### Operation Sequence
1. Validates that index is within valid range (0 to elementCount-1)
2. Validates that element size matches buffer element size (if element.diSize > 0)
3. Copies the element at the specified index to the output parameter
4. Shifts all elements after the index one position to the left using MEMMOVE
5. Clears the last position (now empty after the shift)
6. Decrements the element count

### Use Cases
```iecst
VAR
    buffer : AnyBuffer;
    value : DINT;
END_VAR

// Remove element from middle of buffer
buffer.PushRight(100);  // [100]
buffer.PushRight(200);  // [100, 200]
buffer.PushRight(300);  // [100, 200, 300]
buffer.PopAtIndex(1, value);  // value = 200, buffer = [100, 300]
```

### Performance Considerations
- **Time complexity**: O(n) - requires shifting elements after the index
- **Memory operations**: One memcpy for retrieval, one MEMMOVE for shifting, one memset for clearing
- **Cost varies by index**:
  - PopAtIndex(0) is equivalent to PopLeft - shifts all remaining elements
  - PopAtIndex(elementCount-1) is equivalent to PopRight - no shifting needed
  - Middle indices require partial shifting
- Use PopRight for O(1) removal when index doesn't matter
- Use for priority queues or sorted list maintenance

### Return Value
- **TRUE**: Element was successfully popped from the specified index
- **FALSE**: Pop operation failed (see error conditions)

### Error Conditions
- Returns FALSE and logs error if index is out of bounds (< 0 or >= elementCount)
- Returns FALSE and logs error if buffer is empty (elementCount = 0)
- Returns FALSE and logs error if element size doesn't match buffer element size (when element.diSize > 0)
- Element parameter can have diSize = 0 to discard the value without copying

### Side Effects
- Shifts all elements after the index one position to the left
- Clears the last element position (sets to zero)
- Decrements bufferMetadata.elementCount by 1

### Dependencies
- Uses memcpy for element retrieval
- Uses MEMMOVE for shifting elements (handles overlapping memory)
- Uses memset for clearing the last position
- Uses Trace for error logging

### Comparison with Other Methods
- **PopAtIndex(0)**: Same as PopLeft - removes from front, shifts all - O(n)
- **PopAtIndex(elementCount-1)**: Same as PopRight - removes from back, no shift - O(1)
- **PopAtIndex(middle)**: Removes from middle, shifts elements after index - O(n)
- **DeleteAtIndex**: Removes without retrieving value - O(1) for last index, O(n) otherwise

### Unittests
 - PopFromBeginning : verify popping at index 0 retrieves first element and shifts all
 - PopFromMiddle : verify popping from middle index retrieves correct element and shifts remaining
 - PopFromEnd : verify popping at last index (elementCount-1) retrieves last element
 - ReturnsTrueOnSuccess : verify method returns TRUE when pop succeeds
 - ReturnsFalseOnNegativeIndex : verify FALSE returned for negative index
 - ReturnsFalseOnIndexOutOfBounds : verify FALSE returned when index >= elementCount
 - ReturnsFalseOnEmptyBuffer : verify FALSE returned when buffer is empty (elementCount = 0)
 - WrongElementSize : verify FALSE returned when element size doesn't match
 - EmptyElement : verify behavior when element.diSize is 0 (discard mode)
 - ShiftsElementsCorrectly : verify all elements after index shift left by one position
 - ClearsLastPosition : verify the last position is cleared to zero after shift
 - DecrementsElementCount : verify elementCount decreases by 1 after pop
 - ConsecutivePops : verify multiple consecutive PopAtIndex calls maintain correct state
 - PopAllElements : verify can pop all elements sequentially using index 0
 - ElementOrderPreserved : verify element order is preserved after pop (except removed element)
 - PopAtIndexEquivalentToPopLeft : verify PopAtIndex(0) behaves same as PopLeft
 - PopAtIndexEquivalentToPopRight : verify PopAtIndex(elementCount-1) behaves same as PopRight
*)
PopAtIndex := FALSE;
// Check index bounds, cannot pop what is not filled in
IF index < bufferConfiguration.bufferBoundLower OR index >= bufferConfiguration.bufferBoundLower + bufferMetadata.elementCount THEN
	Trace.Error(__POUNAME(), CONCAT('Pop attempt at invalid index ', TO_STRING(index)));
	RETURN;
END_IF

// Check if buffer is empty
IF isEmpty THEN
	Trace.Error(__POUNAME(), 'Pop attempt on empty buffer');
	RETURN;
END_IF

// rebasedIndex necessary if LL <> 0
rebasedIndex := index - bufferConfiguration.bufferBoundLower;
// TRUE: passed type is not checked, element is discarded and not returned
IF NOT popDiscard THEN
	// Check element size if copy is requested (element.diSize > 0)
	IF element.diSize <> bufferConfiguration.elementSize THEN
		Trace.Error(__POUNAME(), CONCAT('Element size mismatch: expected ', CONCAT(TO_STRING(bufferConfiguration.elementSize), CONCAT(', got ', TO_STRING(element.diSize)))));
		RETURN;
	END_IF

	offset	 := rebasedIndex * bufferConfiguration.elementSize;
	destAddr := element.pValue;
	srcAddr	 := ADR(pBuffer.pValue[offset]);
	nBytes	 := TO_UDINT(element.diSize);
	memcpy(destAddr, srcAddr, nBytes);
END_IF

// Calculate how many elements need to be shifted
elementsToShift := bufferMetadata.elementCount - rebasedIndex - 1;
// Shift elements after the index one position to the left (if any)
IF elementsToShift > 0 THEN
	offset	 := rebasedIndex * bufferConfiguration.elementSize;
	destAddr := ADR(pBuffer.pValue[offset]);								   // destination: current index
	srcAddr	 := ADR(pBuffer.pValue[offset + bufferConfiguration.elementSize]); // source: next index
	nBytes	 := TO_UDINT(elementsToShift * bufferConfiguration.elementSize);
	MEMMOVE(destAddr, srcAddr, nBytes);
END_IF

// Delete last element data 
DeleteAtIndex(bufferMetadata.elementCount + bufferConfiguration.bufferBoundLower - 1);

// Update internal element counters 
CountDecrement();
PopAtIndex := TRUE;
END_METHOD

// Removes and retrieves the first element from the buffer (FIFO/queue operation)
METHOD PopLeft : BOOL
VAR_INPUT
	element	   : ANY;			// Variable to receive the popped element
	popDiscard : BOOL := FALSE; // When TRUE, element is removed but not copied (type checking skipped)
END_VAR

VAR
	offset	 : DINT;
	destAddr : PVOID;
	srcAddr	 : PVOID;
	nBytes	 : UDINT;
END_VAR

(*
## Detailed Description

Removes the first element from the left side of the buffer and optionally copies it to
the provided element parameter. This implements a standard FIFO (First-In-First-Out)
queue operation where elements are dequeued from the front.

The `popDiscard` parameter controls whether the removed element is copied to the output
parameter or simply discarded. This is useful for circular buffer scenarios where you need
to remove elements to make space without retrieving their values.

### Operation Sequence

**When popDiscard = FALSE (default - retrieve element):**
1. Validates that the buffer contains at least one element
2. Validates that element size matches the buffer's configured element size
3. Copies the first element to the output parameter
4. Shifts all remaining elements one position to the left
5. Clears the last position (now empty after the shift)
6. Decrements the element count

**When popDiscard = TRUE (discard element):**
1. Validates that the buffer contains at least one element
2. **Skips element size validation** (type checking bypassed)
3. **Skips copying element** to output parameter
4. Shifts all remaining elements one position to the left
5. Clears the last position (now empty after the shift)
6. Decrements the element count

### Parameters
- **element**: Variable to receive the popped element
  - When popDiscard=FALSE: Must match buffer's element size, receives the popped value
  - When popDiscard=TRUE: Can be any type/size, value is not copied (ignored)
- **popDiscard**: Controls whether to copy element or discard it
  - **FALSE (default)**: Element is validated and copied to output parameter
  - **TRUE**: Element validation is skipped, value is discarded (not copied)
  - Use TRUE for circular buffer overwrite scenarios where you don't need the old value

### Key Features
- **FIFO behavior**: Elements are removed in the order they were added (when combined with PushRight)
- **Optional discard mode**: Can remove element without retrieving it (popDiscard=TRUE)
- **Automatic shifting**: Maintains contiguous element storage after removal
- **Size validation**: Ensures the output element size matches buffer element size (when popDiscard=FALSE)
- **Type safety bypass**: popDiscard=TRUE skips type checking for performance in discard scenarios
- **Safe empty check**: Returns FALSE and logs error if buffer is empty

### Usage Example
```iecst
VAR
    queue : AnyBuffer(pBuffer := myBuffer, bufferBoundLower := 0, bufferBoundUpper := 9, isBufferPersistent := FALSE);
    value : DINT;
    discardBuffer : BYTE;  // Can be any type when using popDiscard=TRUE
    success : BOOL;
END_VAR

// Standard: Pop and retrieve the first element
success := queue.PopLeft(value, FALSE);  // or just queue.PopLeft(value)
IF success THEN
    // Process the retrieved value
END_IF

// Discard mode: Pop without retrieving (e.g., circular buffer overwrite)
success := queue.PopLeft(discardBuffer, TRUE);  // Element removed, value not copied
// OR with temporary pointer-based buffer:
pTemp := __NEW(BYTE, elementSize);
success := queue.PopLeft(pTemp^, TRUE);  // Element removed, discarded to temp buffer
__DELETE(pTemp);
```

### Performance Considerations
- **Time complexity**: O(n) due to element shifting (n = elementCount)
- **Memory operations**: Uses MEMMOVE for efficient bulk memory shifting
- **popDiscard=TRUE**: Slightly faster than popDiscard=FALSE (skips size check and memcpy)
- For frequent left-side operations, consider if a circular buffer would be more efficient

### Return Value
- **TRUE**: Element was successfully popped (and copied if popDiscard=FALSE)
- **FALSE**: Pop operation failed (see error conditions)

### Error Conditions
- Returns FALSE and logs error if buffer is empty (elementCount <= 0)
- Returns FALSE and logs error if element size doesn't match buffer element size **when popDiscard=FALSE**
- When popDiscard=TRUE, element size validation is skipped (no error for size mismatch)

### Dependencies
- Calls DeleteAtIndex to decrement element count and clear the vacated position
- Uses memcpy for element retrieval
- Uses MEMMOVE for shifting elements (handles overlapping memory correctly)
- Uses Trace for error logging

### Unittests
 - RetrievesFirstElement : verify the first element value is copied to output element when popDiscard=FALSE
 - ShiftsElements : verify all elements shift left by one position after pop
 - ClearsLastElement : verify the last position is cleared to zero after shift
 - DecrementsElementCount : verify elementCount decreases by 1 after pop
 - ReturnsTrueOnSuccess : verify method returns TRUE when pop succeeds
 - WrongSize : verify FALSE returned when element size differs from buffer element size (popDiscard=FALSE)
 - EmptyElement : verify behavior when element.diSize is 0 (discard mode, shift only)
 - PopFromEmptyBuffer : verify behavior when buffer has no elements (elementCount = 0)
 - PopSingleElement : verify popping when buffer contains exactly one element
 - ConsecutivePops : verify multiple sequential pops maintain correct order and state
 - PopAfterPushLeft : verify LIFO behavior with PushLeft and PopLeft
 - PopAfterPushRight : verify FIFO behavior with PushRight and PopLeft
 - PopUntilEmpty : verify popping all elements until buffer is empty
 - ElementOrderPreserved : verify remaining elements shift correctly and maintain relative order
 - PopDiscardTrue : verify element is removed but not copied when popDiscard=TRUE
 - PopDiscardTrueSkipsTypeCheck : verify no error when element size is wrong and popDiscard=TRUE
 - PopDiscardTrueShiftsElements : verify elements still shift correctly when popDiscard=TRUE
 - PopDiscardTrueDecrementsCount : verify elementCount decreases when popDiscard=TRUE
 - PopDiscardFalseRetrievesValue : verify element value is copied when popDiscard=FALSE (default)
 - PopDiscardFalseValidatesType : verify type checking occurs when popDiscard=FALSE
 - PopDiscardWithWrongTypeSucceeds : verify PopLeft with wrong type succeeds when popDiscard=TRUE
 - PopDiscardReturnsTrueOnSuccess : verify method returns TRUE when popDiscard=TRUE succeeds
*)
PopLeft := FALSE;
// Check if buffer has elements to pop
IF bufferMetadata.elementCount <= 0 THEN
	Trace.Error(__POUNAME(), 'Cannot pop from empty buffer');
	RETURN;
END_IF

// TRUE: passed type is not checked, element is discarded and not returned
IF NOT popDiscard THEN
	// Check element size if copy is requested (element.diSize > 0)
	IF element.diSize <> bufferConfiguration.elementSize THEN
		Trace.Error(__POUNAME(), CONCAT('Element size mismatch: expected ', CONCAT(TO_STRING(bufferConfiguration.elementSize), CONCAT(', got ', TO_STRING(element.diSize)))));
		RETURN;
	END_IF

	destAddr := element.pValue;
	srcAddr	 := pBuffer.pValue;
	nBytes	 := TO_UDINT(element.diSize);
	memcpy(destAddr, srcAddr, nBytes);
END_IF

// Shift elements to the left
offset	 := bufferConfiguration.elementSize;
destAddr := pBuffer.pValue;
srcAddr	 := ADR(pBuffer.pValue[offset]);
nBytes	 := TO_UDINT((bufferMetadata.elementCount - 1) * bufferConfiguration.elementSize);
MEMMOVE(destAddr, srcAddr, nBytes);

// Delete last element data 
DeleteAtIndex(bufferConfiguration.bufferBoundLower + bufferMetadata.elementCount - 1);

// Update internal element counters 
CountDecrement();
PopLeft := TRUE;
END_METHOD

// Removes and retrieves the last element from the buffer (stack pop operation)
METHOD PopRight : BOOL
VAR_INPUT
	element	   : ANY;			// Variable to receive the popped element
	popDiscard : BOOL := FALSE; // When TRUE, element is removed but not copied (type checking skipped)
END_VAR

VAR
	offset	 : DINT;
	destAddr : PVOID;
	srcAddr	 : PVOID;
	nBytes	 : UDINT;
END_VAR

(*
## Detailed Description

Removes the last element from the right side (back) of the buffer and optionally copies it to
the provided element parameter. This implements a standard stack pop operation where elements
are removed from the back, which can be combined with PushRight for LIFO (Last-In-First-Out)
behavior.

The `popDiscard` parameter controls whether the removed element is copied to the output
parameter or simply discarded. This is useful for circular buffer scenarios where you need
to remove elements to make space without retrieving their values.

### Operation Sequence

**When popDiscard = FALSE (default - retrieve element):**
1. Validates that the buffer contains at least one element
2. Validates that element size matches the buffer's configured element size
3. Copies the last element (at index elementCount-1) to the output parameter
4. Clears the last element position using DeleteAtIndex
5. Decrements the element count
6. No shifting of other elements required

**When popDiscard = TRUE (discard element):**
1. Validates that the buffer contains at least one element
2. **Skips element size validation** (type checking bypassed)
3. **Skips copying element** to output parameter
4. Clears the last element position using DeleteAtIndex
5. Decrements the element count
6. No shifting of other elements required

### Parameters
- **element**: Variable to receive the popped element
  - When popDiscard=FALSE: Must match buffer's element size, receives the popped value
  - When popDiscard=TRUE: Can be any type/size, value is not copied (ignored)
- **popDiscard**: Controls whether to copy element or discard it
  - **FALSE (default)**: Element is validated and copied to output parameter
  - **TRUE**: Element validation is skipped, value is discarded (not copied)
  - Use TRUE for circular buffer overwrite scenarios where you don't need the old value

### Key Features
- **LIFO behavior**: When combined with PushRight, provides stack behavior (last appended is first popped)
- **FIFO behavior**: When combined with PushLeft, provides queue behavior (first appended is last popped)
- **No shifting required**: Direct removal from the end without moving other elements
- **O(1) time complexity**: Constant time operation (much faster than PopLeft)
- **Optional discard mode**: Can remove element without retrieving it (popDiscard=TRUE)
- **Size validation**: Ensures the output element size matches buffer element size (when popDiscard=FALSE)
- **Type safety bypass**: popDiscard=TRUE skips type checking for performance in discard scenarios
- **Safe empty check**: Returns FALSE and logs error if buffer is empty

### Usage Example
```iecst
VAR
    stack : AnyBuffer(pBuffer := myBuffer, bufferBoundLower := 0, bufferBoundUpper := 9, isBufferPersistent := FALSE);
    value : DINT;
    discardBuffer : BYTE;  // Can be any type when using popDiscard=TRUE
    success : BOOL;
END_VAR

// Standard: Pop and retrieve the last element
success := stack.PopRight(value, FALSE);  // or just stack.PopRight(value)
IF success THEN
    // Process the retrieved value
END_IF

// Discard mode: Pop without retrieving (e.g., circular buffer overwrite)
success := stack.PopRight(discardBuffer, TRUE);  // Element removed, value not copied

// LIFO pattern: Last appended is first popped
stack.PushRight(1);  // [1]
stack.PushRight(2);  // [1, 2]
stack.PushRight(3);  // [1, 2, 3]
stack.PopRight(value); // value = 3, buffer = [1, 2]
```

### Performance Considerations
- **Time complexity**: O(1) - constant time operation (no shifting required)
- **Memory operations**: Single memcpy for element retrieval (when popDiscard=FALSE), memset for clearing
- **popDiscard=TRUE**: Slightly faster than popDiscard=FALSE (skips size check and memcpy)
- **Optimal for stack operations**: Use PushRight + PopRight for efficient LIFO stack
- Much faster than PopLeft since no element shifting is needed
- Preferred method for stack-based data structures

### Return Value
- **TRUE**: Element was successfully popped (and copied if popDiscard=FALSE)
- **FALSE**: Pop operation failed (see error conditions)

### Error Conditions
- Returns FALSE and logs error if buffer is empty (elementCount <= 0)
- Returns FALSE and logs error if element size doesn't match buffer element size **when popDiscard=FALSE**
- When popDiscard=TRUE, element size validation is skipped (no error for size mismatch)

### Side Effects
- Clears the last element position (sets to zero)
- Decrements bufferMetadata.elementCount by 1
- No other elements are moved or modified

### Dependencies
- Calls DeleteAtIndex to decrement element count and clear the position
- Uses memcpy for element retrieval
- Uses Trace for error logging

### Comparison with Other Methods
- **PopRight**: Removes from back (index elementCount-1), no shifting - O(1)
- **PopLeft**: Removes from front (index 0), shifts left - O(n)
- **PushRight**: Adds at back, no shifting - O(1)
- **PushLeft**: Adds at front, shifts right - O(n)

### Unittests
 - RetrievesLastElement : verify the last element value is copied to output element when popDiscard=FALSE
 - DoesNotShiftElements : verify no elements are shifted after pop
 - ClearsLastElement : verify the last position is cleared to zero after pop
 - DecrementsElementCount : verify elementCount decreases by 1 after pop
 - ReturnsTrueOnSuccess : verify method returns TRUE when pop succeeds
 - WrongSize : verify FALSE returned when element size differs from buffer element size (popDiscard=FALSE)
 - EmptyElement : verify behavior when element.diSize is 0 (discard mode, no copy)
 - PopFromEmptyBuffer : verify behavior when buffer has no elements (elementCount = 0)
 - PopSingleElement : verify popping when buffer contains exactly one element
 - ConsecutivePops : verify multiple sequential pops maintain correct order and state
 - PopAfterPushRight : verify LIFO behavior with PushRight and PopRight
 - PopAfterPushLeft : verify FIFO behavior with PushLeft and PopRight
 - PopUntilEmpty : verify popping all elements until buffer is empty
 - ElementOrderPreserved : verify remaining elements stay in their original positions
 - PopDiscardTrue : verify element is removed but not copied when popDiscard=TRUE
 - PopDiscardTrueSkipsTypeCheck : verify no error when element size is wrong and popDiscard=TRUE
 - PopDiscardTrueNoShift : verify no element shifting occurs when popDiscard=TRUE (same as default)
 - PopDiscardTrueDecrementsCount : verify elementCount decreases when popDiscard=TRUE
 - PopDiscardFalseRetrievesValue : verify element value is copied when popDiscard=FALSE (default)
 - PopDiscardFalseValidatesType : verify type checking occurs when popDiscard=FALSE
 - PopDiscardWithWrongTypeSucceeds : verify PopRight with wrong type succeeds when popDiscard=TRUE
 - PopDiscardReturnsTrueOnSuccess : verify method returns TRUE when popDiscard=TRUE succeeds
*)
PopRight := FALSE;
// Check if buffer has elements to pop
IF bufferMetadata.elementCount <= 0 THEN
	Trace.Error(__POUNAME(), 'Cannot pop from empty buffer');
	RETURN;
END_IF

// TRUE: passed type is not checked, element is discarded and not returned
IF NOT popDiscard THEN
	// Check element size if copy is requested (element.diSize > 0)
	IF element.diSize <> bufferConfiguration.elementSize THEN
		Trace.Error(__POUNAME(), CONCAT('Element size mismatch: expected ', CONCAT(TO_STRING(bufferConfiguration.elementSize), CONCAT(', got ', TO_STRING(element.diSize)))));
		RETURN;
	END_IF

	// Calculate offset to last element (elementCount - 1)
	offset	 := (bufferMetadata.elementCount - 1) * bufferConfiguration.elementSize;
	destAddr := element.pValue;
	srcAddr	 := ADR(pBuffer.pValue[offset]);
	nBytes	 := TO_UDINT(element.diSize);
	memcpy(destAddr, srcAddr, nBytes);
END_IF

// Delete last element data 
DeleteAtIndex(bufferConfiguration.bufferBoundLower + bufferMetadata.elementCount - 1);

// Update internal element counters 
CountDecrement();
PopRight := TRUE;
END_METHOD

// Insert an element at a specific index, shifting remaining elements right
METHOD PushAtIndex : BOOL
VAR_INPUT
	index	: DINT;
	element : ANY;
END_VAR

VAR
	offset			: DINT;
	destAddr		: PVOID;
	srcAddr			: PVOID;
	nBytes			: UDINT;
	elementsToShift : DINT;
	rebasedIndex	: DINT;
END_VAR

(*
## Detailed Description

Inserts a new element at the specified index by shifting all elements from that index onward
one position to the right, then placing the new element at the specified position. This provides
random-access insertion capability, allowing elements to be added at any position in the buffer
while maintaining contiguous storage.

### Operation Sequence
1. Validates that the buffer has been properly initialized
2. Checks that the buffer has space available (elementCount < capacity)
3. Validates that index is within valid range (0 to elementCount, inclusive)
4. Validates that the element size matches the buffer's configured element size
5. Shifts all elements from index onward one position to the right using MEMMOVE
6. Copies the new element to the specified index position
7. Increments the element count

### Use Cases
```iecst
VAR
    buffer : AnyBuffer;
    value : DINT;
END_VAR

// Insert at various positions
buffer.PushRight(100);  // [100]
buffer.PushRight(300);  // [100, 300]

value := 200;
buffer.PushAtIndex(1, value);  // [100, 200, 300] - inserted 200 between 100 and 300

value := 50;
buffer.PushAtIndex(0, value);  // [50, 100, 200, 300] - inserted 50 at beginning

value := 400;
buffer.PushAtIndex(4, value);  // [50, 100, 200, 300, 400] - inserted 400 at end
```

### Performance Considerations
- **Time complexity**: O(n) - requires shifting elements after the index
- **Memory operations**: One MEMMOVE for shifting, one memcpy for insertion
- **Cost varies by index**:
  - PushAtIndex(0) is equivalent to PushLeft - shifts all elements
  - PushAtIndex(elementCount) is equivalent to PushRight - no shifting needed
  - Middle indices require partial shifting
- Use PushRight for O(1) insertion when order doesn't matter
- Use for maintaining sorted order or priority queue operations

### Return Value
- **TRUE**: Element was successfully inserted at the specified index
- **FALSE**: Insert operation failed (see error conditions)

### Error Conditions
- Returns FALSE and logs error if buffer is not initialized
- Returns FALSE and logs error if buffer is full (elementCount >= capacity)
- Returns FALSE and logs error if index is out of bounds (< 0 or > elementCount)
- Returns FALSE and logs error if element size doesn't match buffer element size
- Note: index = elementCount is valid (append at end)

### Side Effects
- Shifts all elements from index onward one position to the right
- Increments bufferMetadata.elementCount by 1
- New element is placed at the specified index
- All elements at index and beyond move to index+1, index+2, etc.

### Dependencies
- Requires buffer to be initialized via FB_init or Initialize method
- Uses memcpy for element copying
- Uses MEMMOVE for shifting elements (handles overlapping memory correctly)
- Uses Trace for error logging

### Comparison with Other Methods
- **PushAtIndex(0)**: Same as PushLeft - shifts all, adds at front - O(n)
- **PushAtIndex(elementCount)**: Same as PushRight - no shift, adds at end - O(1)
- **PushAtIndex(middle)**: Inserts at middle, shifts elements after index - O(n)
- **PushLeft**: Always inserts at 0 - O(n)
- **PushRight**: Always inserts at end - O(1)

### Unittests
 - InsertAtBeginning : verify inserting at index 0 shifts all elements and inserts at front
 - InsertInMiddle : verify inserting at middle index shifts remaining elements correctly
 - InsertAtEnd : verify inserting at index elementCount appends at end (like PushRight)
 - InsertIntoEmptyBuffer : verify inserting at index 0 in empty buffer works
 - ReturnsTrueOnSuccess : verify method returns TRUE when insert succeeds
 - ReturnsFalseOnNegativeIndex : verify FALSE returned for negative index
 - ReturnsFalseOnIndexOutOfBounds : verify FALSE returned when index > elementCount
 - ReturnsFalseOnFullBuffer : verify FALSE returned when buffer is at capacity
 - WrongElementSize : verify FALSE returned when element size doesn't match
 - IncrementsElementCount : verify elementCount increases by 1 after insert
 - ShiftsElementsCorrectly : verify all elements from index onward shift right by one
 - PreservesElementOrder : verify element order is preserved after insert
 - MultipleInsertions : verify sequential insertions at different indices work correctly
 - InsertAllValidPositions : verify can insert at every valid position (0 to elementCount)
 - PushAtIndexEquivalentToPushLeft : verify PushAtIndex(0) behaves same as PushLeft
 - PushAtIndexEquivalentToPushRight : verify PushAtIndex(elementCount) behaves same as PushRight
*)
PushAtIndex := FALSE;
// Check if buffer has space available
IF isFull THEN
	Trace.Error(__POUNAME(), 'Cannot insert into full buffer');
	RETURN;
END_IF

// Check index bounds (0 to elementCount is valid - can insert at end)
IF index < bufferConfiguration.bufferBoundLower OR index > bufferConfiguration.bufferBoundLower + bufferMetadata.elementCount THEN
	Trace.Error(__POUNAME(), CONCAT('Insert attempt at invalid index ', TO_STRING(index)));
	RETURN;
END_IF

// Check if buffer is initialized
IF NOT isInitialized THEN
	Trace.Error(__POUNAME(), 'Buffer was not properly initialized before inserting');
	RETURN;
END_IF

// Validate element size matches buffer element size
IF element.diSize <> bufferConfiguration.elementSize THEN
	Trace.Error(__POUNAME(), 'Passed element to insert is of improper size');
	RETURN;
END_IF

// rebasedIndex necessary if LL <> 0
rebasedIndex := index - bufferConfiguration.bufferBoundLower;

// Calculate how many elements need to be shifted
elementsToShift := bufferMetadata.elementCount - rebasedIndex;
// Shift elements from index onward one position to the right (if any)
IF elementsToShift > 0 THEN
	offset	 := rebasedIndex * bufferConfiguration.elementSize;
	destAddr := ADR(pBuffer.pValue[offset + bufferConfiguration.elementSize]); // destination: index+1
	srcAddr	 := ADR(pBuffer.pValue[offset]);								   // source: current index
	nBytes	 := TO_UDINT(elementsToShift * bufferConfiguration.elementSize);
	MEMMOVE(destAddr, srcAddr, nBytes);
END_IF

// Copy the new element to the specified index position
offset	 := rebasedIndex * bufferConfiguration.elementSize;
destAddr := ADR(pBuffer.pValue[offset]);
srcAddr	 := element.pValue;
nBytes	 := TO_UDINT(element.diSize);
memcpy(destAddr, srcAddr, nBytes);

// Update internal element counters 
CountIncrement();
PushAtIndex := TRUE;
END_METHOD

// Appends a new element to the left side of the buffer (LIFO/stack push operation)
METHOD PushLeft : BOOL
VAR_INPUT
	element : ANY;
END_VAR

VAR
	offset	 : DINT;
	destAddr : PVOID;
	srcAddr	 : PVOID;
	nBytes	 : UDINT;
END_VAR

(*
## Detailed Description

Appends a new element to the left side (front) of the buffer by shifting all existing
elements one position to the right and inserting the new element at position 0. This
implements a stack-like push operation at the front, which can be combined with PopLeft
for LIFO (Last-In-First-Out) behavior.

### Operation Sequence
1. Validates that the buffer has been properly initialized
2. Checks that the buffer has space available (elementCount < capacity)
3. Validates that the element size matches the buffer's configured element size
4. Shifts all existing elements one position to the right using MEMMOVE
5. Copies the new element to position 0 (leftmost position)
6. Increments the element count

### Key Features
- **LIFO capability**: When combined with PopLeft, provides stack behavior (last appended is first popped)
- **FIFO capability**: When combined with PopRight, provides queue behavior (first appended is last popped)
- **Automatic shifting**: Maintains element contiguity by shifting existing elements right
- **Size validation**: Ensures the input element size matches buffer element size
- **Capacity checking**: Prevents buffer overflow by validating available space
- **Safe operation**: Validates initialization and capacity before modification

### Usage Example
```iecst
VAR
    stack : AnyBuffer(pBuffer := myBuffer, bufferBoundLower := 0, bufferBoundUpper := 9, isBufferPersistent := FALSE);
    value : DINT := 42;
    success : BOOL;
END_VAR

// Append element to the left (front)
success := stack.PushLeft(value);
IF success THEN
    // Element is now at position 0
    // All previous elements shifted right by one position
END_IF

// LIFO pattern: Last appended is first popped
stack.PushLeft(1);  // [1]
stack.PushLeft(2);  // [2, 1]
stack.PushLeft(3);  // [3, 2, 1]
stack.PopLeft(value); // value = 3, buffer = [2, 1]
```

### Performance Considerations
- **Time complexity**: O(n) due to element shifting (n = elementCount)
- **Memory operations**: Uses MEMMOVE for efficient bulk memory shifting
- **Shift overhead**: Every append requires shifting all existing elements
- For frequent left-side operations, consider if a circular buffer would be more efficient
- Use PopLeft with PushLeft for stack behavior (LIFO)
- Use PopRight with PushLeft for queue behavior (FIFO from right)

### Return Value
- **TRUE**: Element was successfully appended to the left side
- **FALSE**: Append operation failed (see error conditions)

### Error Conditions
- Returns FALSE and logs error if buffer is not initialized
- Returns FALSE and logs error if buffer is full (elementCount >= capacity)
- Returns FALSE and logs error if element size doesn't match buffer element size
- All errors are traced via the Trace system for debugging

### Side Effects
- Shifts all existing elements one position to the right
- Increments bufferMetadata.elementCount by 1
- New element is placed at index 0 (leftmost position)
- Previous element at index 0 moves to index 1, etc.

### Dependencies
- Requires buffer to be initialized via FB_init or Initialize method
- Uses memcpy for element copying
- Uses MEMMOVE for shifting elements (handles overlapping memory correctly)
- Uses Trace for error logging

### Comparison with Other Methods
- **PushLeft**: Adds at front (index 0), shifts right - O(n)
- **PopLeft**: Removes from front, shifts left - O(n)
- **PopRight**: Removes from back, no shifting - O(1)
- **PushAtIndex**: Adds at specific position - O(n)

### Unittests
 - AppendsToEmptyBuffer : verify element is inserted at position 0 in empty buffer
 - AppendsToNonEmptyBuffer : verify element is inserted at position 0 and existing elements shift right
 - IncrementsElementCount : verify elementCount increases by 1 after append
 - ShiftsExistingElements : verify all existing elements shift right by one position
 - ReturnsTrueOnSuccess : verify method returns TRUE when append succeeds
 - ReturnsFalseOnFullBuffer : verify method returns FALSE when buffer is at capacity
 - ReturnsFalseOnWrongSize : verify FALSE returned when element size doesn't match buffer element size
 - PreservesExistingData : verify existing element values remain unchanged after shift
 - AppendMultipleElements : verify consecutive appends work correctly (LIFO order)
 - AppendToFullBufferMinus1 : verify append succeeds when buffer has exactly 1 space remaining
 - AppendWhenFullCapacity : verify append fails when elementCount equals capacity
 - AppendZeroSizedElement : verify behavior when element.diSize is 0
 - AppendWithDifferentDataTypes : verify append works with various data types (DINT, REAL, struct)
 - ConsecutivePushAndPopLeft : verify LIFO behavior with alternating PushLeft and PopLeft calls
 - ConsecutivePushAndPopRight : verify FIFO behavior with alternating PushLeft and PopRight calls
 - ElementOrderAfterMultipleAppends : verify element order is correct after multiple appends
 - FillBufferCompletely : verify filling buffer to full capacity works correctly
*)
PushLeft := FALSE;
// Check if buffer has space available
IF isFull THEN
	Trace.Error(__POUNAME(), 'Cannot append to full buffer');
	RETURN;
END_IF

// Check if buffer is initialized
IF NOT isInitialized THEN
	Trace.Error(__POUNAME(), 'Buffer was not properly initialized before appending');
	RETURN;
END_IF

// Check element size if copy is requested (element.diSize > 0)
IF element.diSize <> bufferConfiguration.elementSize THEN
	Trace.Error(__POUNAME(), CONCAT('Element size mismatch: expected ', CONCAT(TO_STRING(bufferConfiguration.elementSize), CONCAT(', got ', TO_STRING(element.diSize)))));
	RETURN;
END_IF

// Shift all existing elements to the right to make room at position 0
destAddr := ADR(pBuffer.pValue[bufferConfiguration.elementSize]); // Start at position 1
srcAddr	 := pBuffer.pValue;										  // Start at position 0
nBytes	 := TO_UDINT(bufferMetadata.elementCount * bufferConfiguration.elementSize);
MEMMOVE(destAddr, srcAddr, nBytes);

// Copy the new element to position 0 (leftmost position)
destAddr := pBuffer.pValue;
srcAddr	 := element.pValue;
nBytes	 := TO_UDINT(element.diSize);
memcpy(destAddr, srcAddr, nBytes);

// Update internal element counters 
CountIncrement();
PushLeft := TRUE;
END_METHOD

// Appends a new element to the right side of the buffer (FIFO/queue enqueue operation)
METHOD PushRight : BOOL
VAR_INPUT
	element : ANY;
END_VAR

VAR
	offset	 : DINT;
	destAddr : PVOID;
	srcAddr	 : PVOID;
	nBytes	 : UDINT;
END_VAR

(*
## Detailed Description

Appends a new element to the right side (back) of the buffer by placing the element at
the next available position (index = elementCount). This implements a standard queue
enqueue operation where elements are added to the back, which can be combined with PopLeft
for FIFO (First-In-First-Out) behavior.

### Operation Sequence
1. Validates that the buffer has been properly initialized
2. Checks that the buffer has space available (elementCount < capacity)
3. Validates that the element size matches the buffer's configured element size
4. Copies the new element to position elementCount (rightmost available position)
5. Increments the element count

### Key Features
- **FIFO capability**: When combined with PopLeft, provides queue behavior (first appended is first popped)
- **LIFO capability**: When combined with PopRight, provides stack behavior (last appended is first popped)
- **No shifting required**: Direct placement at the end without moving existing elements
- **Size validation**: Ensures the input element size matches buffer element size
- **Capacity checking**: Prevents buffer overflow by validating available space
- **Safe operation**: Validates initialization and capacity before modification

### Usage Example
```iecst
VAR
    queue : AnyBuffer(pBuffer := myBuffer, bufferBoundLower := 0, bufferBoundUpper := 9, isBufferPersistent := FALSE);
    value : DINT := 42;
    success : BOOL;
END_VAR

// Append element to the right (back)
success := queue.PushRight(value);
IF success THEN
    // Element is now at position elementCount-1
    // No existing elements are moved
END_IF

// FIFO pattern: First appended is first popped
queue.PushRight(1);  // [1]
queue.PushRight(2);  // [1, 2]
queue.PushRight(3);  // [1, 2, 3]
queue.PopLeft(value);  // value = 1, buffer = [2, 3]
```

### Performance Considerations
- **Time complexity**: O(1) - constant time operation (no shifting required)
- **Memory operations**: Single memcpy for the new element
- **Optimal for queue operations**: Use PushRight + PopLeft for efficient FIFO queue
- Much faster than PushLeft since no element shifting is needed
- Preferred method for building up a buffer sequentially

### Return Value
- **TRUE**: Element was successfully appended to the right side
- **FALSE**: Append operation failed (see error conditions)

### Error Conditions
- Returns FALSE and logs error if buffer is not initialized
- Returns FALSE and logs error if buffer is full (elementCount >= capacity)
- Returns FALSE and logs error if element size doesn't match buffer element size
- All errors are traced via the Trace system for debugging

### Side Effects
- New element is placed at index elementCount (rightmost available position)
- Increments bufferMetadata.elementCount by 1
- No existing elements are moved or modified

### Dependencies
- Requires buffer to be initialized via FB_init or Initialize method
- Uses memcpy for element copying
- Uses Trace for error logging

### Comparison with Other Methods
- **PushRight**: Adds at back (index elementCount), no shifting - O(1)
- **PushLeft**: Adds at front (index 0), shifts right - O(n)
- **PopLeft**: Removes from front, shifts left - O(n)
- **PopRight**: Removes from back, no shifting - O(1)

### Unittests
 - AppendsToEmptyBuffer : verify element is inserted at position 0 in empty buffer
 - AppendsToNonEmptyBuffer : verify element is inserted at position elementCount and no elements shift
 - IncrementsElementCount : verify elementCount increases by 1 after append
 - DoesNotShiftElements : verify no existing elements are moved after append
 - ReturnsTrueOnSuccess : verify method returns TRUE when append succeeds
 - ReturnsFalseOnFullBuffer : verify method returns FALSE when buffer is at capacity
 - ReturnsFalseOnWrongSize : verify FALSE returned when element size doesn't match buffer element size
 - PreservesExistingData : verify existing element values remain unchanged
 - AppendMultipleElements : verify consecutive appends work correctly (FIFO order with PopLeft)
 - AppendToFullBufferMinus1 : verify append succeeds when buffer has exactly 1 space remaining
 - AppendWhenFullCapacity : verify append fails when elementCount equals capacity
 - AppendZeroSizedElement : verify behavior when element.diSize is 0
 - AppendWithDifferentDataTypes : verify append works with various data types (DINT, REAL, struct)
 - ConsecutivePushAndPopLeft : verify FIFO behavior with PushRight and PopLeft calls
 - ConsecutivePushAndPopRight : verify LIFO behavior with PushRight and PopRight calls
 - ElementOrderAfterMultipleAppends : verify element order is correct after multiple appends
 - FillBufferCompletely : verify filling buffer to full capacity works correctly
*)
PushRight := FALSE;
// Check if buffer has space available
IF isFull THEN
	Trace.Error(__POUNAME(), 'Cannot append to full buffer');
	RETURN;
END_IF

// Check if buffer is initialized
IF NOT isInitialized THEN
	Trace.Error(__POUNAME(), 'Buffer was not properly initialized before appending');
	RETURN;
END_IF

// Check element size if copy is requested (element.diSize > 0)
IF element.diSize <> bufferConfiguration.elementSize THEN
	Trace.Error(__POUNAME(), CONCAT('Element size mismatch: expected ', CONCAT(TO_STRING(bufferConfiguration.elementSize), CONCAT(', got ', TO_STRING(element.diSize)))));
	RETURN;
END_IF

// Copy the new element to position elementCount (rightmost available position)
offset	 := bufferMetadata.elementCount * bufferConfiguration.elementSize;
destAddr := ADR(pBuffer.pValue[offset]);
srcAddr	 := element.pValue;
nBytes	 := TO_UDINT(element.diSize);
memcpy(destAddr, srcAddr, nBytes);

// Update internal element counters 
CountIncrement();
PushRight := TRUE;
END_METHOD

// Overwrite an element at a specific index without changing buffer structure or the buffer counters
METHOD ReplaceAtIndex : BOOL
VAR_INPUT
	index	: DINT;
	element : ANY;
END_VAR

VAR
	offset		 : DINT;
	destAddr	 : PVOID;
	srcAddr		 : PVOID;
	nBytes		 : UDINT;
	rebasedIndex : DINT;
END_VAR

(*
## Detailed Description

Overwrites the element at the specified index with a new value without modifying the buffer
metadata or structure. This is a low-level primitive operation that replaces data in-place
without any shifting, insertion, deletion, or metadata updates. The caller is responsible
for validating buffer state if needed.

### Operation Sequence
1. Validates that index is within valid range (0 to capacity-1)
2. Validates that element size matches buffer element size (if element.diSize > 0)
3. Overwrites the element at the specified index with the new value
4. Returns without modifying element count or other elements

### Use Cases
```iecst
VAR
    buffer : AnyBuffer;
    value : DINT;
END_VAR

// Update specific positions (regardless of whether they're "filled")
value := 999;
buffer.ReplaceAtIndex(2, value);  // Overwrites position 2 with 999
// Works even if position 2 was not previously "filled" in logical sense
```

### Performance Considerations
- **Time complexity**: O(1) - constant time operation (direct indexed access)
- **Memory operations**: Single memcpy to overwrite element
- **No buffer modifications**: No shifting, no count changes, no state checking
- **In-place update**: Efficient for updating data at any buffer position
- Optimal for direct memory updates without overhead
- Use for low-level buffer manipulation or custom buffer management

### Return Value
- **TRUE**: Element was successfully replaced at the specified index
- **FALSE**: Replace operation failed (see error conditions)

### Error Conditions
- Returns FALSE and logs error if index is out of bounds (< 0 or >= capacity)
- Returns FALSE and logs error if element size doesn't match buffer element size (when element.diSize > 0)
- Element parameter can have diSize = 0 to skip replacement (returns TRUE if index valid)

### Side Effects
- **Minimal** - Only the element at the specified index is modified
- **Does NOT** modify elementCount or any other metadata
- **Does NOT** check if position is logically "filled" or if buffer is empty
- All other elements remain in their original positions with original values
- No memory allocation or deallocation

### Important Notes
- **No metadata changes**: Does NOT modify elementCount or validate buffer state
- **Caller responsibility**: Calling code must validate buffer state if needed
- **No state checking**: Works at any index within capacity, regardless of elementCount
- **Index range**: Valid indices are [0, capacity-1], not [0, elementCount-1]
- **Low-level primitive**: Designed for internal use or custom buffer management

### Dependencies
- Uses memcpy for element overwriting
- Uses Trace for error logging

### Comparison with Other Methods
- **ReplaceAtIndex**: Updates element at index - O(1), no metadata change
- **PopAtIndex**: Removes element at index - O(n), shifts and updates count
- **PeekAtIndex**: Reads element at index - O(1), validates elementCount
- **DeleteAtIndex**: Clears element - O(1), no metadata change

### Unittests
 - ReplaceAtBeginning : verify replacing at index 0 updates first element correctly
 - ReplaceInMiddle : verify replacing at middle index updates correct element
 - ReplaceAtEnd : verify replacing at last capacity index updates last element
 - ReturnsTrueOnSuccess : verify method returns TRUE when replace succeeds
 - ReturnsFalseOnNegativeIndex : verify FALSE returned for negative index
 - ReturnsFalseOnIndexAtCapacity : verify FALSE returned when index == capacity
 - ReturnsFalseOnIndexAboveCapacity : verify FALSE returned when index > capacity
 - WrongElementSize : verify FALSE returned when element size doesn't match
 - BufferUnchangedExceptIndex : verify all other elements remain unchanged after replace
 - MetadataUnchanged : verify elementCount and all metadata remain unchanged after replace
 - MultipleReplacements : verify sequential replacements at different indices work correctly
 - ReplaceAllCapacityPositions : verify can replace every capacity position (0 to capacity-1)
 - ReplaceWithDifferentValues : verify replace works with various data values
 - ReplaceSameIndexMultipleTimes : verify can overwrite same position repeatedly
 - ReplaceEmptyPosition : verify can replace position that was never filled (elementCount < index < capacity)
 - ReplaceWhenBufferEmpty : verify replace succeeds even when elementCount = 0 (if index < capacity)
*)
ReplaceAtIndex := FALSE;
// Check index bounds against capacity (caller manages state validation)
IF index < bufferConfiguration.bufferBoundLower OR index > bufferConfiguration.bufferBoundUpper THEN
	Trace.Error(__POUNAME(), CONCAT('Replace attempt at invalid index ', TO_STRING(index)));
	RETURN;
END_IF

// Check element size if copy is requested (element.diSize > 0)
IF element.diSize <> bufferConfiguration.elementSize THEN
	Trace.Error(__POUNAME(), CONCAT('Element size mismatch: expected ', CONCAT(TO_STRING(bufferConfiguration.elementSize), CONCAT(', got ', TO_STRING(element.diSize)))));
	RETURN;
END_IF

// rebasedIndex necessary if LL <> 0
rebasedIndex := index - bufferConfiguration.bufferBoundLower;

// Copy element at index to output parameter (if element.diSize > 0)
offset	 := rebasedIndex * bufferConfiguration.elementSize;
destAddr := ADR(pBuffer.pValue[offset]);
srcAddr	 := element.pValue;
nBytes	 := TO_UDINT(element.diSize);
memcpy(destAddr, srcAddr, nBytes);

// No buffer modifications - overwrite-only operation
ReplaceAtIndex := TRUE;
END_METHOD

END_FUNCTION_BLOCK

// Utilities/AnyBuffer/TypedBuffers/LifoBuffer
// Provides a simplified LIFO stack interface as an adapter over AnyBuffer
FUNCTION_BLOCK LifoBuffer IMPLEMENTS I_AnyBufferStrategy
VAR
	anyBuffer	  : I_AnyBuffer;
	isInitialized : BOOL := FALSE;
	_overwrite	  : BOOL := FALSE; // When TRUE, Push overwrites oldest element when full
	_reversed	  : BOOL := FALSE; // When TRUE, reverses push/pop direction (PushLeft/PopLeft)
	{attribute 'hide'}
	discardObject : BYTE; // element for discarding elements in overwrite mode
END_VAR

(*
## Detailed Description

LifoBuffer is an adapter (also known as a strategy or facade) that wraps an AnyBuffer instance
to provide a simplified Last-In-First-Out (LIFO) stack interface. Instead of using the full
AnyBuffer API with directional operations (PushLeft/Right, PopLeft/Right), users can simply
Push and Pop elements following standard stack semantics.

### Alternative Names
In computer science, LIFO data structures are commonly called "Stacks". This implementation
could alternatively be named "Stack" or "StackAdapter" for more conventional naming.

### Design Pattern
This implements the **Adapter Pattern** (also Strategy Pattern), which:
- Wraps a more complex interface (I_AnyBuffer) with a simpler, domain-specific interface
- Delegates all operations to the underlying AnyBuffer instance
- Provides semantic clarity: Push/Pop vs PushRight/PopRight
- Allows multiple strategy implementations (FIFO, LIFO, Priority, etc.) over the same buffer

### LIFO Semantics
- **Push(element)**: Adds element using PushRight (reversed=FALSE) or PushLeft (reversed=TRUE)
- **Pop(element)**: Removes element using PopRight (reversed=FALSE) or PopLeft (reversed=TRUE)
- Push and Pop operate on the **same end** of the buffer (unlike FIFO)
- Last element pushed is the first element popped (LIFO behavior)
- Elements maintain insertion order, but retrieval is in reverse order

### Configurable Behavior
The LifoBuffer supports two optional parameters during initialization:

**overwrite parameter:**
- **FALSE (default)**: Push fails when buffer is full, returns FALSE and logs error
- **TRUE**: Push to full buffer automatically removes element to make space (circular buffer behavior)
  - When reversed=FALSE: Removes from front (PopLeft), adds to back (PushRight)
  - When reversed=TRUE: Removes from back (PopRight), adds to front (PushLeft)
  - Removed element is discarded using internal temporary buffer

**reversed parameter:**
- **FALSE (default)**: Standard LIFO - Push to back (PushRight), Pop from back (PopRight)
- **TRUE**: Reversed direction - Push to front (PushLeft), Pop from front (PopLeft)
- Both Push and Pop operate on the **same end** to maintain LIFO semantics

### Operation Mapping
**Standard Mode (overwrite=FALSE, reversed=FALSE):**
```
Push()  -> anyBuffer.PushRight()  // Add to back (right)
Pop()   -> anyBuffer.PopRight()   // Remove from back (right) - LIFO
Clear() -> anyBuffer.Clear()      // Clear all
isEmpty -> anyBuffer.isEmpty      // Check if empty
isFull  -> anyBuffer.isFull       // Check if full
```

**Overwrite Mode (overwrite=TRUE, reversed=FALSE):**
```
Push()  -> if full: anyBuffer.PopLeft(pBufferTemp), then anyBuffer.PushRight()
Pop()   -> anyBuffer.PopRight()   // Remove from back (right)
```

**Reversed Mode (overwrite=FALSE, reversed=TRUE):**
```
Push()  -> anyBuffer.PushLeft()   // Add to front (left)
Pop()   -> anyBuffer.PopLeft()    // Remove from front (left) - LIFO
```

**Overwrite + Reversed Mode (overwrite=TRUE, reversed=TRUE):**
```
Push()  -> if full: anyBuffer.PopRight(pBufferTemp), then anyBuffer.PushLeft()
Pop()   -> anyBuffer.PopLeft()    // Remove from front (left)
```

### Usage Examples

**Standard LIFO Mode (Stack):**
```iecst
VAR
    rawBuffer : ARRAY[0..2] OF DINT;
    buffer : AnyBuffer(pBuffer := rawBuffer,
                       bufferBoundLower := 0,
                       bufferBoundUpper := 2,
                       isBufferPersistent := FALSE);
    lifo : LifoBuffer(anyBuffer := buffer, overwrite := FALSE, reversed := FALSE);
    value : DINT;
END_VAR

// Push elements (adds to back)
value := 100; lifo.Push(value);  // Stack: [100]
value := 200; lifo.Push(value);  // Stack: [100, 200] - 200 added to back
value := 300; lifo.Push(value);  // Stack: [100, 200, 300] - 300 added to back

// Pop elements (LIFO order - newest first)
lifo.Pop(value);   // value = 300 (from back), Stack: [100, 200]
lifo.Pop(value);   // value = 200 (from back), Stack: [100]
lifo.Pop(value);   // value = 100 (from back), Stack: []
```

**Overwrite Mode (Circular Stack):**
```iecst
VAR
    lifo : LifoBuffer(anyBuffer := buffer, overwrite := TRUE, reversed := FALSE);
END_VAR

// Fill buffer
value := 100; lifo.Push(value);  // Stack: [100]
value := 200; lifo.Push(value);  // Stack: [100, 200]
value := 300; lifo.Push(value);  // Stack: [100, 200, 300]

// Push to full buffer overwrites oldest (from opposite end)
value := 400; lifo.Push(value);  // Stack: [200, 300, 400] - 100 was removed from front
value := 500; lifo.Push(value);  // Stack: [300, 400, 500] - 200 was removed from front
```

**Reversed Mode (reversed=TRUE):**
```iecst
VAR
    lifo : LifoBuffer(anyBuffer := buffer, overwrite := FALSE, reversed := TRUE);
END_VAR

// Push elements (adds to front using PushLeft)
value := 100; lifo.Push(value);  // Stack: [100]
value := 200; lifo.Push(value);  // Stack: [200, 100] - 200 added to front
value := 300; lifo.Push(value);  // Stack: [300, 200, 100] - 300 added to front

// Pop elements (removes from front using PopLeft - LIFO)
lifo.Pop(value);   // value = 300 (from front), Stack: [200, 100]
lifo.Pop(value);   // value = 200 (from front), Stack: [100]
lifo.Pop(value);   // value = 100 (from front), Stack: []
```

### Advantages
- **Simplified interface**: Push/Pop instead of PushRight/PopRight
- **Semantic clarity**: Code intention is clearer with stack terminology
- **Flexibility**: Easy to swap different buffer strategies (FIFO, LIFO, etc.)
- **Type safety**: Enforces LIFO semantics at compile time through interface

### Limitations
- No random access: Cannot peek at arbitrary indices (use AnyBuffer directly if needed)
- No priority queue: Elements are strictly LIFO ordered
- Overwrite mode loses oldest data when buffer is full (from opposite end)
- Combining overwrite and reversed modes creates a circular stack operating from opposite end

### Dependencies
- Requires I_AnyBuffer implementation (e.g., AnyBuffer)
- Uses Trace for error logging and verbose diagnostics
- Implements I_AnyBufferStrategy interface

### Related Patterns
- **FifoBuffer**: Implements queue (First-In-First-Out) semantics
- **PriorityBuffer**: Would implement priority queue with ordered insertion
- **CircularBuffer**: Would implement ring buffer with overwrite semantics
*)

// Removes all elements from the stack and resets to empty state
METHOD Clear : BOOL

(*
## Detailed Description

Clears all elements from the underlying buffer, resetting it to an empty state.
After calling Clear, isEmpty will return TRUE and elementCount will be 0.

This operation delegates directly to the underlying anyBuffer.Clear() method.

### Return Value
- **TRUE**: Stack was successfully cleared
- **FALSE**: Clear operation failed (e.g., anyBuffer is not initialized)

### Side Effects
- All elements are removed from the buffer
- Element count is reset to 0
- Buffer capacity is restored to maximum
- Logs verbose trace message on success
*)
Clear := FALSE;
IF anyBuffer <> 0 THEN
	Clear := anyBuffer.Clear();
	;
END_IF

Trace.Verbose(__POUNAME(), 'executed');
END_METHOD

// Initializes the LIFO stack by injecting the underlying buffer dependency
METHOD FB_Init : BOOL
VAR_INPUT
	bInitRetains : BOOL;		// TRUE: the retain variables are initialized (reset warm / reset cold)
	bInCopyCode	 : BOOL;		// TRUE: the instance will be copied to the copy code afterward (online change)
	anyBuffer	 : I_AnyBuffer; // The underlying buffer implementation to wrap
	overwrite	 : BOOL;		// When TRUE, Push overwrites oldest element when full
	reversed	 : BOOL;		// When TRUE, reverses push/pop direction (PushLeft/PopLeft)
END_VAR

(*
## Detailed Description

Initializes the LifoBuffer by injecting the underlying AnyBuffer dependency. This follows
the dependency injection pattern where the buffer implementation is provided during
construction rather than being created internally.

### Initialization Sequence
1. Validates that a valid anyBuffer reference is provided (non-zero pointer)
2. Stores the buffer reference for use by Push, Pop, and other operations
3. Allocates temporary buffer for discarding elements in overwrite mode
4. Sets isInitialized flag to TRUE to enable operations

### Parameters
- **anyBuffer**: Reference to an I_AnyBuffer implementation (e.g., AnyBuffer instance)
  - Must be a valid, initialized buffer
  - This LifoBuffer will delegate all operations to this buffer
- **overwrite**: Controls behavior when pushing to a full buffer
  - **FALSE (default)**: Push returns FALSE and logs error when buffer is full
  - **TRUE**: Push automatically removes an element from opposite end to make space
    - When reversed=FALSE: Removes from front (PopLeft), adds to back (PushRight)
    - When reversed=TRUE: Removes from back (PopRight), adds to front (PushLeft)
  - Discarded element is popped to internal temporary buffer (pBufferTemp)
- **reversed**: Controls the direction of both Push and Pop operations
  - **FALSE (default)**: Push to back (PushRight), Pop from back (PopRight) - standard stack
  - **TRUE**: Push to front (PushLeft), Pop from front (PopLeft) - reversed stack
  - Both operations work on the **same end** to maintain LIFO semantics

### Return Value
Returns BOOL but value is not evaluated by the runtime. Always call with valid anyBuffer.

### Usage Example
```iecst
VAR
    rawBuffer : ARRAY[0..9] OF DINT;
    buffer : AnyBuffer(pBuffer := rawBuffer,
                       bufferBoundLower := 0,
                       bufferBoundUpper := 9,
                       isBufferPersistent := FALSE);
    lifo : LifoBuffer(anyBuffer := buffer,
                      overwrite := FALSE,
                      reversed := FALSE);
END_VAR
```

### Important Notes
- Must provide a valid anyBuffer reference, otherwise Push/Pop will fail
- The underlying buffer must already be initialized before passing to FB_Init
- A temporary buffer (pBufferTemp) is allocated internally for discarding elements in overwrite mode
- pBufferTemp is automatically deallocated in FB_exit
- Overwrite mode is useful when newest data is more important than oldest
- Reversed mode changes the operational direction of both Push and Pop
- Combining overwrite=TRUE and reversed=TRUE creates a circular stack operating from the opposite end
*)
IF anyBuffer <> 0 THEN
	THIS^.anyBuffer := anyBuffer;
	_overwrite		:= overwrite;
	_reversed		:= reversed;
	isInitialized	:= TRUE;
END_IF
END_METHOD

// Returns TRUE if the stack contains no elements
PROPERTY isEmpty : BOOL

(*
## Detailed Description

Returns TRUE if the stack is empty (contains no elements), FALSE otherwise.
This property delegates directly to the underlying anyBuffer.isEmpty property.

Use this property to check if Pop operation would succeed before attempting to
remove an element.

### Return Value
- **TRUE**: Stack is empty (elementCount = 0)
- **FALSE**: Stack contains one or more elements

### Usage Example
```iecst
IF NOT lifo.isEmpty THEN
    lifo.Pop(value);  // Safe to pop
END_IF
```
*)
GET
isEmpty := anyBuffer.isEmpty;
END_GET
END_PROPERTY

// Returns TRUE if the stack is at maximum capacity
PROPERTY isFull : BOOL

(*
## Detailed Description

Returns TRUE if the stack is full (at maximum capacity), FALSE otherwise.
This property delegates directly to the underlying anyBuffer.isFull property.

Use this property to check if Push operation would succeed before attempting to
add an element.

### Return Value
- **TRUE**: Stack is full (elementCount = capacity)
- **FALSE**: Stack has space for more elements

### Usage Example
```iecst
IF NOT lifo.isFull THEN
    value := 100;
    lifo.Push(value);  // Safe to push
END_IF
```
*)
GET
isFull := anyBuffer.isFull;
END_GET
END_PROPERTY

// Removes and retrieves an element from the stack (LIFO pop operation)
{attribute 'hasanytype'}
METHOD Pop : BOOL
VAR_INPUT
	element : ANY; // Variable to receive the popped element
END_VAR

(*
## Detailed Description

Removes and retrieves an element from the stack. The behavior depends on the 'reversed'
initialization parameter, but always maintains LIFO (Last-In-First-Out) semantics.

**When reversed = FALSE (default mode):**
- Removes element from the back (right side, highest index)
- Delegates to anyBuffer.PopRight()
- Standard stack behavior - last pushed is first popped

**When reversed = TRUE (reversed mode):**
- Removes element from the front (left side, index 0)
- Delegates to anyBuffer.PopLeft()
- Reversed direction but still LIFO - last pushed (to front) is first popped

### Operation Sequence
1. Validates that the buffer has been initialized
2. Validates that element size matches the buffer's configured element size
3. Checks that the stack is not empty
4. Removes element using PopRight (default) or PopLeft (reversed) based on reversed setting
5. Copies the element value to the output parameter
6. For PopLeft: Shifts remaining elements left; For PopRight: No shifting needed
7. Logs verbose trace on success or error trace on failure

### Standard Mode Example (reversed = FALSE)
```iecst
// Push to back, Pop from back (LIFO)
value := 100; lifo.Push(value);  // Stack: [100]
value := 200; lifo.Push(value);  // Stack: [100, 200] - 200 added to back
value := 300; lifo.Push(value);  // Stack: [100, 200, 300] - 300 added to back

lifo.Pop(value);  // Returns 300 (from back), Stack: [100, 200]
lifo.Pop(value);  // Returns 200 (from back), Stack: [100]
lifo.Pop(value);  // Returns 100 (from back), Stack: []
```

### Reversed Mode Example (reversed = TRUE)
```iecst
// Push to front, Pop from front (LIFO)
value := 100; lifo.Push(value);  // Stack: [100]
value := 200; lifo.Push(value);  // Stack: [200, 100] - 200 added to front
value := 300; lifo.Push(value);  // Stack: [300, 200, 100] - 300 added to front

lifo.Pop(value);  // Returns 300 (from front), Stack: [200, 100]
lifo.Pop(value);  // Returns 200 (from front), Stack: [100]
lifo.Pop(value);  // Returns 100 (from front), Stack: []
```

### Return Value
- **TRUE**: Element was successfully popped and copied to element parameter
- **FALSE**: Pop operation failed (see error conditions)

### Error Conditions
- Returns FALSE and logs error if buffer was not initialized
- Returns FALSE and logs error if element size doesn't match buffer element size
- Returns FALSE and logs error if stack is empty (no elements to pop)
- Returns FALSE and logs error if underlying PopLeft or PopRight operation fails

### Parameters
- **element**: Must be a writable variable (not a literal) of the correct size
  - Must match the buffer's configured element size
  - Will receive the popped element value on success

### Side Effects
- Removes one element from the stack
- Decrements element count by 1
- For reversed=FALSE (PopRight): No element shifting required
- For reversed=TRUE (PopLeft): Shifts remaining elements one position to the left
- Logs verbose trace message on success
- Logs error trace message on failure
*)
Pop := FALSE;
IF NOT isInitialized THEN
	Trace.Error(__POUNAME(), 'Buffer was not initialized yet, execute method .init() at least once');
	RETURN;
END_IF

// valid sized element?
IF element.diSize <> anyBuffer.Configuration.elementSize THEN
	Trace.Error(__POUNAME(), 'Passed element to pop to is of improper size');
	RETURN;
END_IF

// retrieve element from buffer if there is any left
IF NOT isEmpty THEN
	IF _reversed THEN
		// Reversed: pop from front (left) - LIFO
		Pop := anyBuffer.PopLeft(element);
	ELSE
		// Standard: pop from back (right) - LIFO
		Pop := anyBuffer.PopRight(element);
	END_IF
ELSE
	Trace.Error(__POUNAME(), 'Attempt to pop from empty buffer');
END_IF

// Pop was ok, trace message
IF Pop THEN
	Trace.Verbose(__POUNAME(), 'executed');
ELSE
	Trace.Error(__POUNAME(), 'FAILED');
END_IF
END_METHOD

// Adds a new element to the stack (LIFO push operation, direction depends on reversed setting)
{attribute 'hasanytype'}
METHOD Push : BOOL
VAR_INPUT
	element : ANY; // Element to add to the stack
END_VAR

(*
## Detailed Description

Adds a new element to the stack. The push direction and overwrite behavior depend on
the 'reversed' and 'overwrite' initialization parameters. Push and Pop operate on the
**same end** of the buffer to maintain LIFO semantics.

**Push Direction (reversed parameter):**
- **reversed = FALSE (default)**: Delegates to anyBuffer.PushRight() - adds to back/right
- **reversed = TRUE**: Delegates to anyBuffer.PushLeft() - adds to front/left

**Overwrite Behavior (overwrite parameter):**
- **overwrite = FALSE (default)**: Push fails if buffer is full, returns FALSE and logs error
- **overwrite = TRUE (circular buffer mode)**: Push succeeds even when buffer is full
  - When reversed=FALSE: Removes element from front (PopLeft to pBufferTemp), then adds to back (PushRight)
  - When reversed=TRUE: Removes element from back (PopRight to pBufferTemp), then adds to front (PushLeft)
  - Discarded element is popped to internal temporary buffer and dropped
  - Useful for scenarios where newest data is more important than oldest

### Operation Sequence

**Standard Mode (overwrite = FALSE, reversed = FALSE):**
1. Validates that the buffer has been initialized
2. Validates that element size matches the buffer's configured element size
3. Checks that the stack is not full (has available capacity)
4. If full: Returns FALSE and logs error
5. If not full: Adds element to the back using PushRight
6. Logs verbose trace on success or error trace on failure

**Standard Mode with Reversed (overwrite = FALSE, reversed = TRUE):**
1. Validates that the buffer has been initialized
2. Validates that element size matches the buffer's configured element size
3. Checks that the stack is not full (has available capacity)
4. If full: Returns FALSE and logs error
5. If not full: Adds element to the front using PushLeft
6. Logs verbose trace on success or error trace on failure

**Overwrite Mode (overwrite = TRUE, reversed = FALSE):**
1. Validates that the buffer has been initialized
2. Validates that element size matches the buffer's configured element size
3. If buffer is full: Removes oldest element from front using PopLeft (discards to pBufferTemp)
4. Adds new element to the back using PushRight
5. Logs verbose trace on success or error trace on failure

**Overwrite Mode with Reversed (overwrite = TRUE, reversed = TRUE):**
1. Validates that the buffer has been initialized
2. Validates that element size matches the buffer's configured element size
3. If buffer is full: Removes oldest element from back using PopRight (discards to pBufferTemp)
4. Adds new element to the front using PushLeft
5. Logs verbose trace on success or error trace on failure

### Standard Mode Example (overwrite = FALSE)
```iecst
// Starting with empty stack
value := 100; lifo.Push(value);  // Stack: [100]
value := 200; lifo.Push(value);  // Stack: [100, 200]
value := 300; lifo.Push(value);  // Stack: [100, 200, 300]

// Pop operations retrieve in LIFO order (newest first)
lifo.Pop(value);  // Returns 300 (last pushed)
lifo.Pop(value);  // Returns 200 (second to last)
lifo.Pop(value);  // Returns 100 (first pushed)
```

### Overwrite Mode Example (overwrite = TRUE)
```iecst
// Assuming buffer capacity is 3
value := 100; lifo.Push(value);  // Stack: [100]
value := 200; lifo.Push(value);  // Stack: [100, 200]
value := 300; lifo.Push(value);  // Stack: [100, 200, 300] - full

// Push to full buffer overwrites oldest (from opposite end)
value := 400; lifo.Push(value);  // Stack: [200, 300, 400] - 100 removed from front
value := 500; lifo.Push(value);  // Stack: [300, 400, 500] - 200 removed from front
```

### Return Value
- **TRUE**: Element was successfully pushed to the stack
- **FALSE**: Push operation failed (see error conditions)

### Error Conditions
- Returns FALSE and logs error if buffer was not initialized
- Returns FALSE and logs error if element size doesn't match buffer element size
- Returns FALSE and logs error if stack is full AND overwrite is FALSE
- Returns FALSE and logs error if underlying PushRight or PushLeft operation fails
- In overwrite mode, Push should always succeed unless buffer is not initialized or element size is wrong

### Parameters
- **element**: Must be a writable variable (not a literal) of the correct size
  - Must match the buffer's configured element size
  - Value will be copied into the stack

### Side Effects

**Standard Mode (overwrite = FALSE):**
- Adds one element to the stack
- No shifting of existing elements required (for PushRight)
- Shifts elements right (for PushLeft when reversed=TRUE)
- Increments element count by 1
- Decrements available capacity by 1
- Logs verbose trace message on success
- Logs error trace message on failure

**Overwrite Mode (overwrite = TRUE):**
- If buffer is full: Removes oldest element from opposite end first
- Adds new element to the push end
- Element count remains constant when overwriting
- Logs verbose trace message on success
- Logs error trace message on failure

### Performance Considerations
- **Standard mode (reversed=FALSE)**: O(1) - PushRight is constant time, no shifting
- **Standard mode (reversed=TRUE)**: O(n) - PushLeft requires shifting all elements right
- **Overwrite mode (reversed=FALSE)**: O(n) when full (PopLeft with shifting + PushRight)
- **Overwrite mode (reversed=TRUE)**: O(n) when full (PopRight O(1) + PushLeft O(n))
- **Overwrite mode**: O(1) or O(n) when not full (depends on reversed setting)
- Pop operation with reversed=FALSE has O(1) complexity (PopRight, no shifting)
- Pop operation with reversed=TRUE has O(n) complexity (PopLeft with shifting)
- Trade-off: reversed=FALSE optimizes both Push and Pop, reversed=TRUE makes Push slower
*)
Push := FALSE;
IF NOT isInitialized THEN
	Trace.Error(__POUNAME(), 'Buffer was not initialized yet, execute method .init() at least once');
	RETURN;
END_IF

// valid sized element pushed?
IF element.diSize <> anyBuffer.Configuration.elementSize THEN
	Trace.Error(__POUNAME(), 'Pushed element is of improper size');
	RETURN;
END_IF

// handle full buffer based on overwrite setting
IF isFull THEN
	IF _overwrite THEN
		// Overwrite mode: remove element from opposite end to make space (discard to pBufferTemp)
		IF _reversed THEN
			// Reversed: remove from back before adding to front
			anyBuffer.PopRight(discardObject, TRUE);
		ELSE
			// Standard: remove from front before adding to back
			anyBuffer.PopLeft(discardObject, TRUE);
		END_IF
	ELSE
		// Standard mode: fail and log error
		Trace.Error(__POUNAME(), 'Attempt to push to full buffer');
		RETURN;
	END_IF
END_IF

// add element based on direction setting (same end as Pop for LIFO)
IF _reversed THEN
	// Reversed: add to front (left)
	Push := anyBuffer.PushLeft(element);
ELSE
	// Standard: add to back (right)
	Push := anyBuffer.PushRight(element);
END_IF

// Push was ok, trace message
IF Push THEN
	Trace.Verbose(__POUNAME(), 'executed');
ELSE
	Trace.Error(__POUNAME(), 'FAILED');
END_IF
END_METHOD

END_FUNCTION_BLOCK

// Utilities/AnyBuffer/TypedBuffers/ListBuffer
// Provides a directional FIFO list with automatic shift-and-overwrite when full
FUNCTION_BLOCK ListBuffer IMPLEMENTS I_AnyBufferStrategy
VAR
	anyBuffer	  : I_AnyBuffer;
	isInitialized : BOOL := FALSE;
	_reversed	  : BOOL := FALSE; // TRUE: add at left, FALSE: add at right (end)
END_VAR

(*
## Detailed Description

List is an adapter that wraps an AnyBuffer instance to provide a configurable-direction
FIFO (First-In-First-Out) list with automatic shift-and-overwrite capability. Unlike a
simple ring buffer, this implementation physically shifts elements when the buffer is full
to maintain contiguous storage and consistent indexing.

### Design Rationale
This adapter is called "List" because it provides list-like semantics:
- Elements are stored contiguously in memory
- Insertion direction can be configured (prepend vs append)
- Automatic capacity management with shift-on-overwrite
- Maintains FIFO ordering regardless of fill direction

### Design Pattern
This implements the **Adapter Pattern** with directional configuration:
- Wraps the AnyBuffer interface with configurable list semantics
- Delegates all operations to the underlying AnyBuffer instance
- Provides automatic shift-and-overwrite when buffer reaches capacity
- Uses private helper methods for clean code organization

### Directional Fill Semantics

**Fill From Left (fillFromLeft = TRUE)**:
- Push adds at index 0 (AppendLeft) - newest at front
- Pop removes from highest index (PopRight) - oldest at end
- When full: Remove oldest (PopRight), add new (AppendLeft)
- Visual: [newest] ← [older] ← [oldest]

**Fill From Right (fillFromLeft = FALSE)**:
- Push adds at end (AppendRight) - newest at end
- Pop removes from index 0 (PopLeft) - oldest at front
- When full: Remove oldest (PopLeft), add new (AppendRight)
- Visual: [oldest] → [older] → [newest]

### Operation Mapping

**When fillFromLeft = TRUE:**
```
Push() not full  -> AppendLeft()          // Add to front
Push() full      -> PopRight() + AppendLeft()  // Remove oldest (end), add new (front)
Pop()            -> PopRight()            // Remove oldest (end)
```

**When fillFromLeft = FALSE:**
```
Push() not full  -> AppendRight()         // Add to end
Push() full      -> PopLeft() + AppendRight()  // Remove oldest (front), add new (end)
Pop()            -> PopLeft()             // Remove oldest (front)
```

### Usage Example - Fill From Left

```iecst
VAR
    rawBuffer : ARRAY[0..2] OF DINT;  // 3-element buffer
    buffer : AnyBuffer(pBuffer := rawBuffer,
                       bufferBoundLower := 0,
                       bufferBoundUpper := 2,
                       isBufferPersistent := FALSE);
    list : List(anyBuffer := buffer, fillFromLeft := TRUE);
    value : DINT;
END_VAR

// Fill from left (prepend)
value := 100; list.Push(value);  // Buffer: [100]
value := 200; list.Push(value);  // Buffer: [200, 100]
value := 300; list.Push(value);  // Buffer: [300, 200, 100] - Full

// Push to full buffer - oldest (100) removed, new prepended
value := 400; list.Push(value);  // Buffer: [400, 300, 200]
value := 500; list.Push(value);  // Buffer: [500, 400, 300]

// Pop removes oldest (from end)
list.Pop(value);  // value = 300, Buffer: [500, 400]
list.Pop(value);  // value = 400, Buffer: [500]
```

### Usage Example - Fill From Right

```iecst
VAR
    rawBuffer : ARRAY[0..2] OF DINT;  // 3-element buffer
    buffer : AnyBuffer(pBuffer := rawBuffer,
                       bufferBoundLower := 0,
                       bufferBoundUpper := 2,
                       isBufferPersistent := FALSE);
    list : List(anyBuffer := buffer, fillFromLeft := FALSE);
    value : DINT;
END_VAR

// Fill from right (append)
value := 100; list.Push(value);  // Buffer: [100]
value := 200; list.Push(value);  // Buffer: [100, 200]
value := 300; list.Push(value);  // Buffer: [100, 200, 300] - Full

// Push to full buffer - oldest (100) removed, new appended
value := 400; list.Push(value);  // Buffer: [200, 300, 400]
value := 500; list.Push(value);  // Buffer: [300, 400, 500]

// Pop removes oldest (from front)
list.Pop(value);  // value = 300, Buffer: [400, 500]
list.Pop(value);  // value = 400, Buffer: [500]
```

### Shift-and-Overwrite Visualization (fillFromLeft = FALSE)

```
Initial state (capacity 3):
[ ][ ][ ]

After pushing 100, 200, 300:
[100][200][300]  <- Full
 ↑           ↑
oldest    newest

After pushing 400 (shifts and overwrites):
Step 1: PopLeft removes 100
[200][300][ ]

Step 2: AppendRight adds 400
[200][300][400]
 ↑           ↑
oldest    newest

After pushing 500:
[300][400][500]
 ↑           ↑
oldest    newest
```

### Advantages
- **Consistent indexing**: Elements always occupy contiguous indices starting from 0
- **Configurable direction**: Can optimize for prepend or append patterns
- **Automatic capacity management**: Always maintains most recent N elements
- **Predictable memory layout**: No internal index tracking, uses actual array positions
- **Clean implementation**: Private helper methods separate concerns

### Use Cases
- **Directional data streams**: Logs that grow in specific direction
- **Time-series data**: Keep most recent N samples with natural ordering
- **Event history**: Maintain fixed-size event list with temporal ordering
- **Undo/redo buffers**: Limited-size command history
- **Message queues**: Fixed-size message buffers with FIFO ordering

### Comparison with Other Adapters

| Feature | FifoBuffer | RingBuffer | List |
|---------|-----------|------------|------|
| Overwrite when full | No (fails) | Yes | Yes |
| Fill direction | Fixed | Fixed | Configurable |
| Physical shifting | Always | On overwrite | On overwrite |
| Index stability | No | No | Yes (contiguous) |
| Use case | Queue | Circular log | Directional list |

### Performance Considerations

**Fill From Left (fillFromLeft = TRUE)**:
- **Push (not full)**: O(n) - AppendLeft shifts all elements
- **Push (full)**: O(n) - PopRight + AppendLeft, double shift
- **Pop**: O(1) - PopRight removes last element

**Fill From Right (fillFromLeft = FALSE)**:
- **Push (not full)**: O(1) - AppendRight adds to end
- **Push (full)**: O(n) - PopLeft shifts + AppendRight
- **Pop**: O(n) - PopLeft shifts remaining elements

**Recommendation**: Set fillFromLeft based on your access pattern:
- Frequent pushes, infrequent pops: fillFromLeft = FALSE (O(1) push)
- Frequent pops, infrequent pushes: fillFromLeft = TRUE (O(1) pop)

### Private Helper Methods

The implementation uses private helper methods for code organization:
- `pushInternal()`: Encapsulates push logic with direction handling
- `popInternal()`: Encapsulates pop logic with direction handling
- `removeOldest()`: Removes oldest element based on fill direction

This separation improves:
- Code readability and maintainability
- Testability of individual operations
- Reusability of common logic

### Dependencies
- Requires I_AnyBuffer implementation (e.g., AnyBuffer)
- Uses Trace for error logging and verbose diagnostics
- Implements I_AnyBufferStrategy interface

### Related Patterns
- **FifoBuffer**: FIFO without overwrite, fixed left-to-right fill
- **RingBuffer**: Circular buffer with overwrite, fixed fill direction
- **LifoBuffer**: Stack (Last-In-First-Out) semantics
*)

// Removes all elements from the list and resets to empty state
METHOD Clear : BOOL

(*
## Detailed Description

Clears all elements from the underlying buffer, resetting it to an empty state.
After calling Clear, isEmpty will return TRUE and elementCount will be 0.

This operation delegates directly to the underlying anyBuffer.Clear() method.

### Return Value
- **TRUE**: List was successfully cleared
- **FALSE**: Clear operation failed (e.g., anyBuffer is not initialized)

### Side Effects
- All elements are removed from the buffer
- Element count is reset to 0
- Buffer capacity is restored to maximum
- Logs verbose trace message on success
*)
Clear := FALSE;
IF anyBuffer <> 0 THEN
	Clear := anyBuffer.Clear();
END_IF

Trace.Verbose(__POUNAME(), 'executed');
END_METHOD

// Initializes the list by injecting the underlying buffer dependency
METHOD FB_Init : BOOL
VAR_INPUT
	bInitRetains : BOOL;		  // TRUE: the retain variables are initialized (reset warm / reset cold)
	bInCopyCode	 : BOOL;		  // TRUE: the instance will be copied to the copy code afterward (online change)
	anyBuffer	 : I_AnyBuffer;	  // The underlying buffer implementation to wrap
	fillFromLeft : BOOL := FALSE; // TRUE: fill from left (prepend), FALSE: fill from right (append)
END_VAR

(*
## Detailed Description

Initializes the List by injecting the underlying AnyBuffer dependency and configuring
the fill direction. This follows the dependency injection pattern where the buffer
implementation and behavior are provided during construction.

### Initialization Sequence
1. Validates that a valid anyBuffer reference is provided (non-zero pointer)
2. Stores the buffer reference for use by Push, Pop, and other operations
3. Stores the fillFromLeft flag to control insertion direction
4. Sets isInitialized flag to TRUE to enable operations

### Parameters
- **anyBuffer**: Reference to an I_AnyBuffer implementation (e.g., AnyBuffer instance)
  - Must be a valid, initialized buffer
  - This List will delegate all operations to this buffer
- **fillFromLeft**: Controls insertion direction and FIFO ordering
  - **FALSE** (default): Fill from right - AppendRight for push, PopLeft for pop
    - Newest elements at high indices, oldest at index 0
    - Optimized for frequent pushes (O(1))
  - **TRUE**: Fill from left - AppendLeft for push, PopRight for pop
    - Newest elements at index 0, oldest at high indices
    - Optimized for frequent pops (O(1))

### Return Value
Returns BOOL but value is not evaluated by the runtime. Always call with valid anyBuffer.

### Usage Example - Append Mode (fillFromLeft = FALSE)
```iecst
VAR
    rawBuffer : ARRAY[0..9] OF DINT;
    buffer : AnyBuffer(pBuffer := rawBuffer,
                       bufferBoundLower := 0,
                       bufferBoundUpper := 9,
                       isBufferPersistent := FALSE);
    list : List(anyBuffer := buffer,
                fillFromLeft := FALSE);  // Append mode (default)
END_VAR
// Push is O(1), Pop is O(n)
```

### Usage Example - Prepend Mode (fillFromLeft = TRUE)
```iecst
VAR
    rawBuffer : ARRAY[0..9] OF DINT;
    buffer : AnyBuffer(pBuffer := rawBuffer,
                       bufferBoundLower := 0,
                       bufferBoundUpper := 9,
                       isBufferPersistent := FALSE);
    list : List(anyBuffer := buffer,
                fillFromLeft := TRUE);  // Prepend mode
END_VAR
// Push is O(n), Pop is O(1)
```

### Important Notes
- Must provide a valid anyBuffer reference, otherwise Push/Pop will fail
- The underlying buffer must already be initialized before passing to FB_Init
- Choose fillFromLeft based on your access pattern for optimal performance
- The fill direction cannot be changed after initialization
*)
IF anyBuffer <> 0 THEN
	THIS^.anyBuffer := anyBuffer;
	THIS^._reversed := fillFromLeft;
	isInitialized	:= TRUE;
END_IF
END_METHOD

// Returns TRUE if the list contains no elements
PROPERTY isEmpty : BOOL

(*
## Detailed Description

Returns TRUE if the list is empty (contains no elements), FALSE otherwise.
This property delegates directly to the underlying anyBuffer.isEmpty property.

Use this property to check if Pop operation would succeed before attempting to
remove an element.

### Return Value
- **TRUE**: List is empty (elementCount = 0)
- **FALSE**: List contains one or more elements

### Usage Example
```iecst
IF NOT list.isEmpty THEN
    list.Pop(value);  // Safe to pop
END_IF
```
*)
GET
isEmpty := anyBuffer.isEmpty;
END_GET
END_PROPERTY

// Returns TRUE if the list is at maximum capacity
PROPERTY isFull : BOOL

(*
## Detailed Description

Returns TRUE if the list is full (at maximum capacity), FALSE otherwise.
This property delegates directly to the underlying anyBuffer.isFull property.

Note: Push will still succeed when isFull is TRUE by automatically removing the
oldest element and shifting remaining elements. This property is informational
and indicates when the next Push will trigger shift-and-overwrite behavior.

### Return Value
- **TRUE**: List is full (elementCount = capacity)
- **FALSE**: List has space for more elements

### Usage Example
```iecst
IF list.isFull THEN
    // Next Push will remove oldest element and shift
    Trace.Info('List', 'Next push will overwrite oldest element');
END_IF

value := 100;
success := list.Push(value);  // Will succeed even if full
```
*)
GET
isFull := anyBuffer.isFull;
END_GET
END_PROPERTY

// Removes and retrieves the oldest element from the list (FIFO dequeue)
{attribute 'hasanytype'}
METHOD Pop : BOOL
VAR_INPUT
	element : ANY; // Variable to receive the popped element
END_VAR

(*
## Detailed Description

Removes and retrieves the oldest element from the list following FIFO (First-In-First-Out)
semantics. The location of the oldest element depends on the fillFromLeft configuration:
- fillFromLeft = TRUE: Oldest at end (highest index), uses PopRight
- fillFromLeft = FALSE: Oldest at front (index 0), uses PopLeft

This method delegates to the private popInternal() helper method for implementation.

### Operation by Fill Direction

**Fill From Left (fillFromLeft = TRUE)**:
- Oldest element is at highest index (end of list)
- Uses PopRight to remove (O(1) operation)
- No shifting required

**Fill From Right (fillFromLeft = FALSE)**:
- Oldest element is at index 0 (front of list)
- Uses PopLeft to remove (O(n) operation)
- All remaining elements shift one position left

### Return Value
- **TRUE**: Element was successfully popped and copied to element parameter
- **FALSE**: Pop operation failed (see error conditions)

### Error Conditions
- Returns FALSE and logs error if buffer was not initialized
- Returns FALSE and logs error if element size doesn't match buffer element size
- Returns FALSE and logs error if list is empty (no elements to pop)
- Returns FALSE and logs error if underlying pop operation fails

### Parameters
- **element**: Must be a writable variable (not a literal) of the correct size
  - Must match the buffer's configured element size
  - Will receive the popped element value on success

### Side Effects
- Removes one element from the list
- May shift remaining elements (fillFromLeft = FALSE)
- Decrements element count by 1
- Increases available capacity by 1
- Logs verbose trace message on success
- Logs error trace message on failure

### Performance
- **fillFromLeft = TRUE**: O(1) - removes from end, no shifting
- **fillFromLeft = FALSE**: O(n) - removes from front, shifts all remaining elements
*)
Pop := FALSE;
IF NOT isInitialized THEN
	Trace.Error(__POUNAME(), 'Buffer was not initialized yet, execute method .init() at least once');
	RETURN;
END_IF

// Valid sized element?
IF element.diSize <> anyBuffer.Configuration.elementSize THEN
	Trace.Error(__POUNAME(), 'Passed element to pop to is of improper size');
	RETURN;
END_IF

// Check if empty
IF isEmpty THEN
	Trace.Error(__POUNAME(), 'Attempt to pop from empty buffer');
	RETURN;
END_IF

// pop element based on fill direction
IF _reversed THEN
	// Fill from left: oldest element is at the end (highest index)
	Pop := anyBuffer.PopRight(element);
ELSE
	// Fill from right: oldest element is at the front (index 0)
	Pop := anyBuffer.PopLeft(element);
END_IF

// Trace result
IF Pop THEN
	Trace.Verbose(__POUNAME(), 'executed');
ELSE
	Trace.Error(__POUNAME(), 'FAILED');
END_IF
END_METHOD

// Adds a new element to the list with automatic shift-and-overwrite when full
{attribute 'hasanytype'}
METHOD Push : BOOL
VAR_INPUT
	element : ANY; // Element to add to the list
END_VAR

(*
## Detailed Description

Adds a new element to the list. The insertion location depends on the fillFromLeft
configuration:
- fillFromLeft = TRUE: Adds at front (index 0) using AppendLeft
- fillFromLeft = FALSE: Adds at end using AppendRight

When the list is full, the oldest element is automatically removed and remaining
elements are shifted to make space for the new element.

### Operation Sequence (Not Full)
1. Validates that the buffer has been initialized
2. Validates that element size matches the buffer's configured element size
3. Adds element based on fill direction:
   - fillFromLeft = TRUE: AppendLeft (insert at index 0, shift existing right)
   - fillFromLeft = FALSE: AppendRight (insert at end)
4. Logs verbose trace on success or error trace on failure

### Operation Sequence (Full)
1. Validates that the buffer has been initialized
2. Validates that element size matches the buffer's configured element size
3. Removes oldest element based on fill direction:
   - fillFromLeft = TRUE: PopRight removes from end
   - fillFromLeft = FALSE: PopLeft removes from front and shifts
4. Adds new element based on fill direction:
   - fillFromLeft = TRUE: AppendLeft adds at front and shifts
   - fillFromLeft = FALSE: AppendRight adds at end
5. Logs verbose trace on success or error trace on failure

### Fill From Left Example (fillFromLeft = TRUE)
```iecst
// Buffer capacity = 3
value := 100; list.Push(value);  // [100]
value := 200; list.Push(value);  // [200, 100]
value := 300; list.Push(value);  // [300, 200, 100] - Full

// Push to full: Remove 100 (end), add 400 (front)
value := 400; list.Push(value);  // [400, 300, 200]

// Visual: [newest=400, 300, oldest=200]
list.Pop(value);  // Returns 200 (oldest from end)
```

### Fill From Right Example (fillFromLeft = FALSE)
```iecst
// Buffer capacity = 3
value := 100; list.Push(value);  // [100]
value := 200; list.Push(value);  // [100, 200]
value := 300; list.Push(value);  // [100, 200, 300] - Full

// Push to full: Remove 100 (front), add 400 (end)
value := 400; list.Push(value);  // [200, 300, 400]

// Visual: [oldest=200, 300, newest=400]
list.Pop(value);  // Returns 200 (oldest from front)
```

### Return Value
- **TRUE**: Element was successfully pushed to the list
- **FALSE**: Push operation failed (see error conditions)

### Error Conditions
- Returns FALSE and logs error if buffer was not initialized
- Returns FALSE and logs error if element size doesn't match buffer element size
- Returns FALSE and logs error if underlying append operation fails

### Parameters
- **element**: Must be a writable variable (not a literal) of the correct size
  - Must match the buffer's configured element size
  - Value will be copied into the list

### Side Effects (Not Full)
- Adds one element to the list
- May shift existing elements (fillFromLeft = TRUE shifts right)
- Increments element count by 1
- Decrements available capacity by 1

### Side Effects (Full)
- Removes oldest element
- Shifts remaining elements (direction depends on fillFromLeft)
- Adds new element
- Element count remains at maximum capacity

### Performance
**fillFromLeft = TRUE (prepend mode)**:
- Not full: O(n) - AppendLeft shifts all existing elements right
- Full: O(n) - PopRight (O(1)) + AppendLeft (O(n))

**fillFromLeft = FALSE (append mode)**:
- Not full: O(1) - AppendRight adds to end
- Full: O(n) - PopLeft (O(n)) + AppendRight (O(1))

Choose fillFromLeft based on your access pattern for optimal performance.
*)
Push := FALSE;
IF NOT isInitialized THEN
	Trace.Error(__POUNAME(), 'Buffer was not initialized yet, execute method .init() at least once');
	RETURN;
END_IF

// Valid sized element?
IF element.diSize <> anyBuffer.Configuration.elementSize THEN
	Trace.Error(__POUNAME(), 'Pushed element is of improper size');
	RETURN;
END_IF

// If buffer is full, remove oldest element first
IF isFull THEN
	IF NOT removeOldest() THEN
		Trace.Error(__POUNAME(), 'Failed to remove oldest element');
		RETURN;
	END_IF
END_IF

// push element based on fill direction
IF _reversed THEN
	// Fill from left: add new element at front (index 0)
	Push := anyBuffer.PushLeft(element);
ELSE
	// Fill from right: add new element at end
	Push := anyBuffer.PushRight(element);
END_IF

// Trace result
IF Push THEN
	Trace.Verbose(__POUNAME(), 'executed');
ELSE
	Trace.Error(__POUNAME(), 'FAILED');
END_IF
END_METHOD

// Private helper method to remove the oldest element based on fill direction
METHOD PRIVATE removeOldest : BOOL
VAR
	dummyElement : ANYTYPE; // For discarding oldest element
END_VAR

(*
## Detailed Description

Private helper method that removes the oldest element from the list based on the
fill direction. This method is called by Push() when the buffer is full to make
space for a new element.

### Operation
- fillFromLeft = TRUE: Oldest at end (high index), uses PopRight
- fillFromLeft = FALSE: Oldest at front (index 0), uses PopLeft

The removed element is discarded as we only care about making space.

### Return Value
- **TRUE**: Oldest element was successfully removed
- **FALSE**: Remove operation failed

### Side Effects
- Removes one element from the list
- May shift remaining elements (fillFromLeft = FALSE)
- Decrements element count by 1
- Increases available capacity by 1
*)
removeOldest := FALSE;
IF _reversed THEN
	// Fill from left: oldest element is at the end (highest index)
	removeOldest := anyBuffer.PopRight(dummyElement, TRUE);
ELSE
	// Fill from right: oldest element is at the front (index 0)
	removeOldest := anyBuffer.PopLeft(dummyElement, TRUE);
END_IF
END_METHOD

END_FUNCTION_BLOCK

// Utilities/AnyBuffer/TypedBuffers/RingBuffer
// Provides a circular buffer (ring buffer) interface with automatic overwrite capability
FUNCTION_BLOCK RingBuffer IMPLEMENTS I_AnyBufferStrategy
VAR
	anyBuffer	  : I_AnyBuffer;
	isInitialized : BOOL := FALSE;
	_overwrite	  : BOOL := TRUE; // TRUE: overwrites oldest when full
END_VAR

(*
## Detailed Description

RingBuffer is an adapter that wraps an AnyBuffer instance to provide circular buffer
(also called ring buffer) semantics with automatic overwrite capability. When the buffer
is full and a new element is added, the oldest element is automatically removed to make
space, creating a continuous circular data flow.

### Alternative Names
This data structure is commonly known as:
- **Ring Buffer**: Emphasizes the circular/wrap-around nature
- **Circular Buffer**: Describes the logical circular structure
- **Cyclic Buffer**: Another term for the same concept

### Design Pattern
This implements the **Adapter Pattern**, which:
- Wraps the AnyBuffer interface with domain-specific circular buffer semantics
- Delegates all operations to the underlying AnyBuffer instance
- Provides automatic overwrite behavior when buffer reaches capacity
- Useful for streaming data, logging, and producer-consumer patterns

### Ring Buffer Semantics
- **Push(element)**: Adds element using circular indexing (FIFO enqueue)
  - When not full: Uses WriteAtIndex for direct write at tail position
  - When full: Overwrites oldest element using WriteAtIndex (no shifting!)
- **Pop(element)**: Removes oldest element using PeekAtIndex and circular head pointer (no shifting!)
- **Automatic overwrite**: When enabled and buffer is full, oldest data is overwritten in place
- **Circular indexing**: Uses head/tail pointers to track logical queue positions
- **Direct memory access**: Uses WriteAtIndex for O(1) writes without counter overhead
- Elements maintain FIFO order (first in, first out)

### Operation Mapping
```
Push() when not full  -> anyBuffer.WriteAtIndex(tail, ...)  // Direct write (O(1), no counter overhead)
Push() when full      -> anyBuffer.WriteAtIndex(tail, ...)  // Overwrite oldest (O(1), no shift!)
Pop()                 -> anyBuffer.PeekAtIndex(head, ...)   // Read oldest (O(1), no shift!)
Clear()               -> anyBuffer.Clear()                  // Clear all + reset indices
isEmpty               -> (elementCount = 0)                 // Check element count
isFull                -> (elementCount >= capacity)         // Check element count
```

### Usage Example
```iecst
VAR
    rawBuffer : ARRAY[0..2] OF DINT;  // Small buffer for demonstration
    buffer : AnyBuffer(pBuffer := rawBuffer,
                       bufferBoundLower := 0,
                       bufferBoundUpper := 2,
                       isBufferPersistent := FALSE);
    ring : RingBuffer(anyBuffer := buffer, overwrite := TRUE);
    value : DINT;
END_VAR

// Fill buffer
value := 100; ring.Push(value);  // Buffer: [100]
value := 200; ring.Push(value);  // Buffer: [100, 200]
value := 300; ring.Push(value);  // Buffer: [100, 200, 300] (full)

// Push to full buffer - oldest (100) is automatically removed
value := 400; ring.Push(value);  // Buffer: [200, 300, 400]
value := 500; ring.Push(value);  // Buffer: [300, 400, 500]

// Pop retrieves in FIFO order
ring.Pop(value);  // value = 300, Buffer: [400, 500]
```

### Circular Buffer Visualization
```
Initial state (capacity 5):
[ ][ ][ ][ ][ ]

After pushing 100, 200, 300:
[100][200][300][ ][ ]

After filling completely (100, 200, 300, 400, 500):
[100][200][300][400][500]  <- Full

After pushing 600 (overwrites 100):
[600][200][300][400][500]
     ^                ^
   oldest          newest

After pushing 700 (overwrites 200):
[600][700][300][400][500]
          ^             ^
       oldest       newest
```

### Advantages
- **No data loss when streaming**: Automatically maintains most recent data
- **Constant memory usage**: Buffer size never grows beyond capacity
- **Highly efficient**: Both Push and Pop are O(1) with circular indexing (no shifting!)
- **Simple interface**: Push/Pop semantics like FifoBuffer
- **Predictable behavior**: Always keeps newest data when overwrite is enabled
- **True circular buffer**: Implements proper ring buffer with head/tail pointers

### Use Cases
- **Logging buffers**: Keep most recent N log messages
- **Sensor data streams**: Store latest readings, discard old data
- **Audio/video buffers**: Maintain continuous data flow
- **Producer-consumer patterns**: Decouple data production and consumption rates
- **History tracking**: Keep fixed-size history of events or states

### Comparison with FifoBuffer
| Feature | FifoBuffer | RingBuffer |
|---------|-----------|------------|
| Behavior when full | Rejects new elements | Overwrites oldest |
| Push operation | Fails if full | Always succeeds |
| Data loss | Never (rejects push) | Yes (by design) |
| Use case | Queue with backpressure | Streaming data |
| Memory | Fixed size | Fixed size |

### Overwrite Behavior
- **overwrite = TRUE**: Push to full buffer removes oldest, adds newest (circular)
- **overwrite = FALSE**: Push to full buffer fails (same as FifoBuffer)

### Limitations
- No random access: Cannot peek at arbitrary indices (use AnyBuffer directly if needed)
- Overwrite is automatic: Cannot prevent data loss when buffer is full (by design)
- No notification: Caller is not informed when overwrite occurs

### Dependencies
- Requires I_AnyBuffer implementation (e.g., AnyBuffer)
- Uses Trace for error logging and verbose diagnostics
- Implements I_AnyBufferStrategy interface

### Performance Considerations
- **Push when not full**: O(1) - uses AppendRight
- **Push when full**: O(1) - uses ReplaceAtIndex with circular indexing (no shifting!)
- **Pop**: O(1) - uses PeekAtIndex with circular indexing (no shifting!)
- **Overall**: True O(1) constant-time operations for all Push and Pop operations
- Ideal for high-performance scenarios with frequent overwrites and streaming data

### Related Patterns
- **FifoBuffer**: FIFO queue without overwrite (rejects when full)
- **LifoBuffer**: Stack (Last-In-First-Out) semantics
- **PriorityBuffer**: Priority queue with ordered insertion
*)

METHOD PRIVATE AdvanceHead
// Advance tail pointer (circular)
anyBuffer.Metadata.headIndex := anyBuffer.Metadata.headIndex + 1;
IF anyBuffer.Metadata.headIndex > anyBuffer.Configuration.bufferBoundUpper THEN
	anyBuffer.Metadata.headIndex := anyBuffer.Configuration.bufferBoundLower;
END_IF
END_METHOD

METHOD PRIVATE AdvanceTail
// Advance tail pointer (circular)
anyBuffer.Metadata.tailIndex := anyBuffer.Metadata.tailIndex + 1;
IF anyBuffer.Metadata.tailIndex > anyBuffer.Configuration.bufferBoundUpper THEN
	anyBuffer.Metadata.tailIndex := anyBuffer.Configuration.bufferBoundLower;
END_IF
END_METHOD

// Removes all elements from the ring buffer and resets to empty state
METHOD Clear : BOOL

(*
## Detailed Description

Clears all elements from the underlying buffer, resetting it to an empty state.
After calling Clear, isEmpty will return TRUE and elementCount will be 0.

This operation delegates directly to the underlying anyBuffer.Clear() method.

### Return Value
- **TRUE**: Ring buffer was successfully cleared
- **FALSE**: Clear operation failed (e.g., anyBuffer is not initialized)

### Side Effects
- All elements are removed from the buffer
- Element count is reset to 0
- Buffer capacity is restored to maximum
- Logs verbose trace message on success
*)
Clear := FALSE;
IF anyBuffer <> 0 THEN
	Clear := anyBuffer.Clear();

	// Reset circular buffer indices
	anyBuffer.Metadata.headIndex	:= anyBuffer.Configuration.bufferBoundLower;
	anyBuffer.Metadata.tailIndex	:= anyBuffer.Configuration.bufferBoundLower;
	anyBuffer.Metadata.elementCount := 0;
END_IF

Trace.Verbose(__POUNAME(), 'executed');
END_METHOD

// Initializes the ring buffer by injecting the underlying buffer dependency
METHOD FB_Init : BOOL
VAR_INPUT
	bInitRetains : BOOL;		 // TRUE: the retain variables are initialized (reset warm / reset cold)
	bInCopyCode	 : BOOL;		 // TRUE: the instance will be copied to the copy code afterward (online change)
	anyBuffer	 : I_AnyBuffer;	 // The underlying buffer implementation to wrap
	overwrite	 : BOOL := TRUE; // TRUE: overwrites oldest element when full (circular behavior)
END_VAR

(*
## Detailed Description

